FUNCTION_BLOCK MockEvent IMPLEMENTS I_Event
VAR
	_name : T_MAXSTRING;
END_VAR

END_FUNCTION_BLOCK

(* stored: Version 1.1.0.1, ProductVersion 3.1.4024.12
   POU MockEvent: Id {92fe7472-59ce-063f-0ff1-2c7ed3de4a75}, SpecialFunc None *)
